{attribute 'linkalways'} 
{attribute 'no_explicit_call' := 'This FB is a CLASS and must be accessed using methods or properties'}
{attribute 'enable_dynamic_creation'}
FUNCTION_BLOCK ResetCommand EXTENDS AxisCommand

METHOD FB_init : BOOL
VAR_INPUT
	bInitRetains : BOOL; // if TRUE, the retain variables are initialized (warm start / cold start)
	bInCopyCode : BOOL;  // if TRUE, the instance afterwards gets moved into the copy code (online change)
	axisRef : REFERENCE TO Axis;
END_VAR
_axisRef REF= axisRef;
END_METHOD

METHOD PROTECTED  WhileBusy
VAR_INPUT
	CommandState : I_CommandBusyState;
END_VAR
VAR_INST
	_fb : MC_Reset;
END_VAR
_fb(
	Axis := _axisRef._InternalAxisRef,
	Execute := TRUE
);

IF _fb.Busy THEN
	RETURN;
END_IF

_fb(Axis := _axisRef._InternalAxisRef, Execute := FALSE);

IF _fb.Error THEN
	CommandState.SetError(_fb.ErrorID);
	RETURN;
END_IF

CommandState.SetDone();
END_METHOD

END_FUNCTION_BLOCK

(* stored: Version 1.1.0.1, ProductVersion 3.1.4024.12
   POU ResetCommand: Id {fbdd2803-8795-42d1-8ee7-9a961a7284c0}, SpecialFunc None
   Folder Constructor: Id {ee8f912a-5352-4190-88f7-9f07ef07cd8a}
   Method FB_init: Id {8faec425-f017-4414-8fa5-d98a0fc8bdd1}
   Method WhileBusy: Id {c12f80ff-11b2-4944-8057-3c7a6478d0e9} *)
